Universal Robots URScript: 00C_01_JieXian_ToYuBei.script

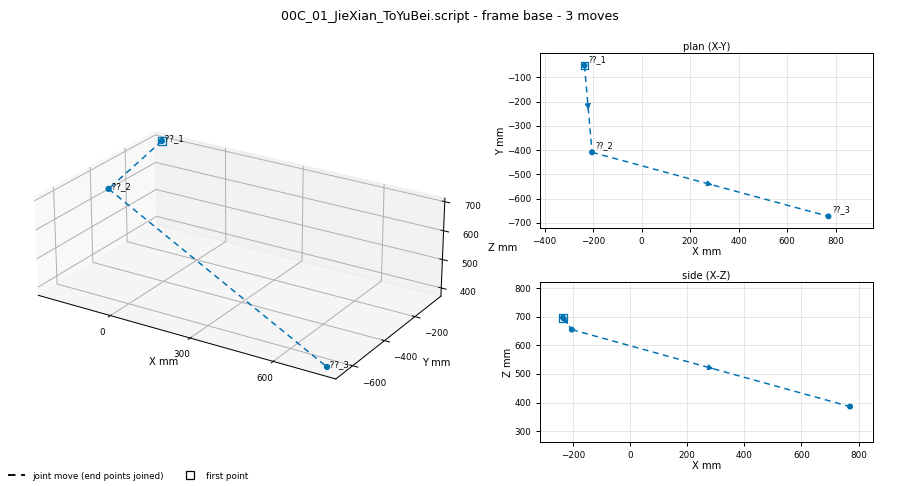
[picture p0: tool path of 00C_01_JieXian_ToYuBei.script in frame base, 3 of 3 moves have a stored position in this frame; points joined in program order, loops and branches not executed]
def P00C_01_JieXian_ToYuBei():
  set_gravity([0.0, 0.0, 9.82])
  set_safety_mode_transition_hardness(1)
  set_standard_analog_input_domain(0, 1)
  set_standard_analog_input_domain(1, 1)
  set_tool_analog_input_domain(0, 1)
  set_tool_analog_input_domain(1, 1)
  set_analog_outputdomain(0, 0)
  set_analog_outputdomain(1, 0)
  set_tool_voltage(24)
  set_input_actions_to_default()
  set_tcp(p[0.0,0.0,0.32,0.0,0.0,-0.5236])
  set_payload(0.0)
  global Zhua_1=[0.08063, -2.42649, -1.72682, -0.47876, 0.40808, -1.10831]
  global prepose=p[0.98979, -0.16931, -0.39963, 1.98720, 0.07234, 0.05469]
  global i_var_2=0
  global i_var_1=True
  global pose=p[0.98979, -0.31931, -0.39963, 1.98720, 0.07234, 0.05469]
  $ 1 "机器人程序"
  $ 2 "MoveJ"
  $ 3 "路点_1"
  set_tcp(p[-0.06262,0.03599,0.32923,0.0,0.0,1.3731])
  movej(get_inverse_kin(p[-.235281377636, -.051146089814, .697573762968, .005856294883, -.018009109240, 1.750391334054], qnear=[-1.5701678434955042, -1.633802997034195E-4, -2.875479523335592, -1.853560749684469, -1.5659878889666956, 0.3726629614830017]), a=0.6981317007977318, v=0.5235987755982988)
  $ 4 "路点_2"
  set_tcp(p[-0.06262,0.03599,0.32923,0.0,0.0,1.3731])
  movej(get_inverse_kin(p[-.204357271349, -.408883540288, .655289716257, .057495987055, -.016371963509, 1.700058523180], qnear=[-1.5328190962420862, -1.589508358632223, -2.6286216417895716, -0.5411513487445276, -1.602502171193258, 0.28854942321777344]), a=0.6981317007977318, v=0.5235987755982988)
  $ 5 "路点_3"
  set_tcp(p[-0.06262,0.03599,0.32923,0.0,0.0,1.3731])
  movej(get_inverse_kin(p[.770170055153, -.672753998243, .385715680602, .061489577452, -.012206245883, 1.533410549624], qnear=[-0.5370209852801722, -2.699575726185934, -1.2693970839129847, -0.7956755797015589, -1.5583208242999476, -0.8679745833026331]), a=0.6981317007977318, v=0.5235987755982988)
end
